// TIA Portal project "one_button_on_off_V17" (V17)

(* hardware
DEVICE "S7-1200 station_1"  S7-1200 Station
   slot 0: "Rack_0"  S7-1200 Rack  Rack  V1.0
   slot 1: "PLC_1"  CPU 1215C DC/DC/DC  6ES7 215-1AG40-0XB0  V4.2
*)

// ===== PLC "PLC_1"  CPU 1215C DC/DC/DC =====

VAR_GLOBAL   // PLC tag table "Default tag table"
   "button" AT %I0.0 : Bool;
   "memory_on" AT %M0.0 : Bool;
   "memory_off" AT %M0.1 : Bool;
   "motor" AT %Q0.0 : Bool;
END_VAR

ORGANIZATION_BLOCK "Main"   // OB1, LAD, ProgramCycle
TITLE = "Main Program Sweep (Cycle)"
{ S7_Optimized_Access := 'TRUE' }
VERSION : 0.1
   VAR_INPUT
      Initial_Call : Bool;   // Initial call of this OB
      Remanence : Bool;   // =True, if remanent data are available
   END_VAR
BEGIN

REGION Network 1
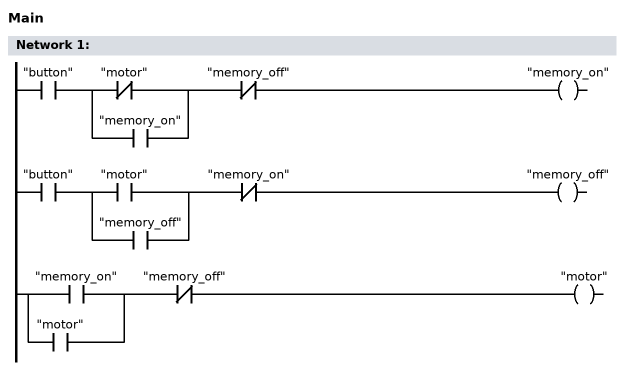
   RUNG wire#powerrail
      Contact( "button" )
      wire#w1
      I_Contact( "motor" )
      wire#w2
      I_Contact( "memory_off" )
      Coil( "memory_on" )
   END_RUNG
   RUNG wire#w1
      Contact( "memory_on" )
   END_RUNG wire#w2
   RUNG wire#powerrail
      Contact( "button" )
      wire#w3
      Contact( "motor" )
      wire#w4
      I_Contact( "memory_on" )
      Coil( "memory_off" )
   END_RUNG
   RUNG wire#w3
      Contact( "memory_off" )
   END_RUNG wire#w4
   RUNG wire#powerrail
      Contact( "memory_on" )
      wire#w5
      I_Contact( "memory_off" )
      Coil( "motor" )
   END_RUNG
   RUNG wire#powerrail
      Contact( "motor" )
   END_RUNG wire#w5
   // the same network as SCL:
   "memory_on" := "button" AND (NOT "motor" OR "memory_on") AND NOT "memory_off";
   "memory_off" := "button" AND ("motor" OR "memory_off") AND NOT "memory_on";
   "motor" := ("memory_on" OR "motor") AND NOT "memory_off";
END_REGION
END_ORGANIZATION_BLOCK